FUNCTION_BLOCK FB_CycleInit
VAR_INPUT
	xStart : BOOL;
END_VAR
VAR_OUTPUT
	fbRtrigStart:R_trig;
	xBusy:BOOL;
	iEtape:INT;
END_VAR
VAR
	fbEtape:FB_Etape;
END_VAR

fbEtape.mActualisation(stParam.stStatus.xModePasAPas,fbBtn.xNextPas);

fbRtrigStart(clk:=fbBtn.xStart);


CASE fbEtape.iNo OF
	0:IF xStart THEN
		fbEtape.piVal:=99;
		END_IF
	99: fbEtape.psMess:='Reset sur les Actionneurs';
		fbEtape.piSVal:=100;
	100:fbEtape.psMess:='Initialiser les positions';
		IF  fbAct1.IxSensIn AND fbAct2.IxSensIn THEN
			fbEtape.piSVal:=999;
		END_IF
	
	999:fbEtape.psMess:='FIN Cycle Init';
		fbEtape.piSVal:=0;
END_CASE

xBusy:=fbEtape.iNo<>0;
iEtape:=fbEtape.iNo;

END_FUNCTION_BLOCK

(* stored: Version 1.1.0.1, ProductVersion 3.1.4020.6
   POU FB_CycleInit: Id {78f8b3c7-c7ef-4e76-a081-037ca3472bc0}, SpecialFunc None *)
